// TC3 retained catalog image, separate from the volatile seed pointer registry.
TYPE ST_LocalRecipeCatalog :
STRUCT
    SchemaVersion : UINT;
    Count : INT;
    Records : ARRAY[1..PL_Fraktal.MAX_RECIPES] OF ST_LocalRecipeRecord;
END_STRUCT
END_TYPE

(* stored: Version 1.1.0.1, ProductVersion 3.1.4024.12
   DUT ST_LocalRecipeCatalog: Id {33f1797a-39e2-47df-9168-489994180277} *)
